FUNCTION_BLOCK PUBLIC MMStatusMonitor
VAR_IN_OUT
	
END_VAR
VAR_INPUT
END_VAR
VAR_OUTPUT
END_VAR
VAR
	HLCStatusTimer		:TON;
	PathStatusTimer		:TON;
	MotorStatusTimer	:TON;
	VehicleStatusTimer	:TON;
	byCounter: BYTE := 1;
	bVehicleJammed: BOOL := FALSE;
	bVehicleLostByMotor: BOOL := FALSE;
	bPrevVehicleJammed : BOOL := FALSE;
	JamTimer :TON;
END_VAR

HLCStatusTimer(IN:=TRUE,PT:=MM_CONST.MM_HLC_STATUS_POLLING);
PathStatusTimer(IN:=TRUE,PT:=MM_CONST.MM_PATH_STATUS_POLLING);
MotorStatusTimer(IN:=TRUE,PT:=MM_CONST.MM_MOTOR_STATUS_POLLING);
VehicleStatusTimer(IN:=TRUE, PT:=MM_CONST.MM_VEHICLE_STATUS_POLLING);

IF (HLCStatusTimer.Q) THEN
		Stations.fbMMSendMsg.M_CmdHLCStatus();
		HLCStatusTimer(IN:=FALSE);
END_IF

IF (PathStatusTimer.Q) THEN
		Stations.fbMMSendMsg.M_CmdHLCStatus(); // to do get path status
		PathStatusTimer(IN:=FALSE);
END_IF

IF (MotorStatusTimer.Q) THEN
		Stations.fbMMSendMsg.M_CmdHLCStatus(); // to do get HLC Status
		MotorStatusTimer(IN:=FALSE);
END_IF

IF (VehicleStatusTimer.Q) THEN
		Stations.fbMMSendMsg.M_CmdVehicleStatus();
		VehicleStatusTimer(IN:=FALSE);
END_IF

bVehicleJammed := FALSE;
bVehicleLostByMotor := FALSE;
FOR byCounter := 1 TO MM_CONST.MAX_VEHICLES BY 1 DO
	bVehicleJammed := bVehicleJammed OR STATUS.MMVehiclesStatus[byCounter].VehicleFlags.2;
	bVehicleLostByMotor := bVehicleLostByMotor OR (STATUS.MMVehiclesStatus[byCounter].VehicleFlags.0 = 0) OR (STATUS.MMVehiclesStatus[byCounter].VehicleFlags.7 = 1);
    STATUS.PartStatusHMI[byCounter] := PartsData.Status[byCounter].OverallStatus;	// this will add color to the vehicles on the HMI
	IF (STATUS.MMVehiclesStatus[byCounter].VehicleFlags.2) THEN STATUS.PartStatusHMI[byCounter] := ePartStatus.eJam; END_IF
END_FOR

IF (bVehicleJammed AND NOT bPrevVehicleJammed) THEN // only when transitioning from non-jammed state to jammed state
	//Stations.fbMMSendMsg.M_CmdSuspendMov();
	//GVL_IO.MM_YEnableMagneMotion := FALSE;
END_IF
bPrevVehicleJammed := bVehicleJammed;  // to ensure that after turning on the MM bus, we don't immediately shut down the MM bus.

IF (bVehicleJammed) THEN JamTimer(IN:=TRUE, PT:=T#40S);
	ELSE 
	JamTimer(IN:=FALSE);
END_IF
IF (GVL_IO.ResumeMovementFromHMI <>0) THEN // Button Click Resume From HMI.
//	Stations.fbMMSendMsg.M_CmdResumeMov();
	GVL_IO.ResumeMovementFromHMI := 0;
	GVL_IO.MM_YEnableMagneMotion := TRUE;
	Stations.fbPrimeMover.ResetPrimeMoverAndPurge(); // this will send prime mover to purrge state
	Stations.fbCycleControl.ResetCycleControlState();

	Stations.fbLoad1Sta.ClearVehicleTrigger();
	Stations.fbLoad2Sta.ClearVehicleTrigger(); 
	Stations.fbLoad3Sta.ClearVehicleTrigger();
	Stations.fbLoad4Sta.ClearVehicleTrigger();
	Stations.fbVisionSta.ClearVehicleTrigger();
	Stations.fbPistonSta.ClearVehicleTrigger();
	Stations.fbCapInsertSta.ClearVehicleTrigger();
	//Stations.fbGoodUnloadSta.ClearVehicleTrigger();
	Stations.fbGoodULSta_1.ClearVehicleTrigger();
	Stations.fbGoodULSta_2.ClearVehicleTrigger();
	Stations.fbGoodULSta_3.ClearVehicleTrigger();
	Stations.fbGoodULSta_4.ClearVehicleTrigger();
	Stations.fbRejectSta.ClearVehicleTrigger();
	Stations.fbIB_StopRobotSta.ClearVehicleTrigger();	
	Stations.fbOB_StopBeforeVisionSta.ClearVehicleTrigger(); 
	Stations.fbOB_StopRobotSta.ClearVehicleTrigger();
	Stations.fbOB_StopRobotSta.MoveToLoading := TRUE;
	
	Stations.fbRoutePlanner.SetRejectLoadPosChoiceToInit();
	Stations.fbRoutePlanner.SetGoodULLoadPosChoiceToInit();
	
	FOR byCounter := 1 TO MM_CONST.MAX_VEHICLES BY 1 DO
			Stations.fbVehicleManager[byCounter].ResetVehicleManager();
	END_FOR	
	
	IF (bVehicleLostByMotor) THEN
		;
	END_IF
END_IF

PROPERTY PUBLIC IsMMJammed : BOOL
GET
IsMMJammed := (JamTimer.Q);
END_GET
SET
END_SET
END_PROPERTY

END_FUNCTION_BLOCK

(* stored: Version 1.1.0.1, ProductVersion 3.1.4022.6
   POU MMStatusMonitor: Id {14f6e4d8-c9ee-4d56-9214-f7809589574d}, SpecialFunc None
   Property IsMMJammed: Id {a26b7db8-39e5-4f0a-b74d-d7a743b31c08}
   Get Get: Id {6ccaea6e-470e-4d2f-b0d2-b75fa81f06e4}
   Set Set: Id {1cb63b9c-4d7d-424c-9107-ac4d899625c8} *)
